(*

## Short summary
This interface provides assert statements for booleans 

.. <legal notes>

legal notes
=================
| SPDX-FileCopyrightText: © 2022 ekvip automation GmbH <info@ekvip.de>
| SPDX-License-Identifier: Apache-2.0
| For details check: Apache-2.0_

.. _Apache-2.0: https://www.apache.org/licenses/LICENSE-2.0

.. </legal notes>



*)

INTERFACE IBooleanAssertion EXTENDS __SYSTEM.IQueryInterface

(*

## Short summary
This assertion method checks if the current value is equal to the expected value

.. <legal notes>

legal notes
=================
| SPDX-FileCopyrightText: © 2022 ekvip automation GmbH <info@ekvip.de>
| SPDX-License-Identifier: Apache-2.0
| For details check: Apache-2.0_

.. _Apache-2.0: https://www.apache.org/licenses/LICENSE-2.0

.. </legal notes>



*)

METHOD valueIsEqualTo
VAR_INPUT
	(* current value to check *)
	currentValue	:BOOL;
	(* expected value to compare *)
	expectedValue	:BOOL;
	(* message if the assertion is false *)
	message			:AssertMessage;
END_VAR
END_METHOD

(*

## Short summary
This assertion method checks if the current value is ``FALSE``

.. <legal notes>

legal notes
=================
| SPDX-FileCopyrightText: © 2022 ekvip automation GmbH <info@ekvip.de>
| SPDX-License-Identifier: Apache-2.0
| For details check: Apache-2.0_

.. _Apache-2.0: https://www.apache.org/licenses/LICENSE-2.0

.. </legal notes>



*)

METHOD valueIsFalse
VAR_INPUT
	(* current value to check *)
	currentValue	:BOOL;
	(* message if the assertion is false *)
	message			:AssertMessage;
END_VAR
END_METHOD

(*

## Short summary
This assertion method checks if the current value is not equal to the unexpected value

.. <legal notes>

legal notes
=================
| SPDX-FileCopyrightText: © 2022 ekvip automation GmbH <info@ekvip.de>
| SPDX-License-Identifier: Apache-2.0
| For details check: Apache-2.0_

.. _Apache-2.0: https://www.apache.org/licenses/LICENSE-2.0

.. </legal notes>



*)

METHOD valueIsNotEqualTo
VAR_INPUT
	(* current value to check *)
	currentValue	:BOOL;
	(* unexpected value to compare *)
	unexpectedValue	:BOOL;
	(* message if the assertion is false *)
	message			:AssertMessage;
END_VAR
END_METHOD

(*

## Short summary
This assertion method checks if the current value is ``TRUE``

.. <legal notes>

legal notes
=================
| SPDX-FileCopyrightText: © 2022 ekvip automation GmbH <info@ekvip.de>
| SPDX-License-Identifier: Apache-2.0
| For details check: Apache-2.0_

.. _Apache-2.0: https://www.apache.org/licenses/LICENSE-2.0

.. </legal notes>



*)

METHOD valueIsTrue
VAR_INPUT
	(* current value to check *)
	currentValue	:BOOL;
	(* message if the assertion is false *)
	message			:AssertMessage;
END_VAR
END_METHOD

END_INTERFACE

(* stored: Version 1.1.0.1, ProductVersion 3.1.4024.11
   Itf IBooleanAssertion: Id {3884a5fe-844d-4647-b096-3f0db78d954b}
   Method valueIsEqualTo: Id {d97fdcf6-7fea-46a4-bea7-2fcb746da995}
   Method valueIsFalse: Id {12de8ec1-514b-4dda-ab01-3f22cf3a4b6c}
   Method valueIsNotEqualTo: Id {5e3bcd93-8617-481b-868f-31a87b02d61c}
   Method valueIsTrue: Id {534edc49-58d7-4ccf-bb09-38b6b8a22337} *)
